Staubli VAL3: padding.pgx

program padding(num x_value1, num x_value2, string& x_return1[], string& x_return2[])
// pad both strings with leading "0" to equal length
  local string l_padding
begin
  call decToBin(roundDown(x_value1),x_return1)
  call decToBin(roundDown(x_value2),x_return2)
  if bDebug
    putln("padding(): "+x_return1+", "+x_return2)
  endIf
  l_padding=""
  call fillStr("0",abs(len(x_return1)-len(x_return2)),l_padding)
  if len(x_return1)<len(x_return2)
    x_return1=l_padding+x_return1
  endIf
  if len(x_return2)<len(x_return1)
    x_return2=l_padding+x_return2
  endIf
  if bDebug
    putln("padding(): "+x_return1+", "+x_return2)
  endIf
end
